FUNCTION_BLOCK FB_TimeLimitedIterator
VAR
    nLocalTaskUsagePercent : BYTE; 
    fbGetTickTime : GETCPUCOUNTER;
    TaskIndex : DINT;
    
    nInterruptThreshold : UDINT;
    nLocalCycleTime : UDINT;
    nIterationStartTime : ULINT;
    nIterationCurrentTime : ULINT;
    nIterationElapsedTime : UDINT;
END_VAR

METHOD PUBLIC CheckInterationTimeExceeded : BOOL
VAR_INPUT
END_VAR
fbGetTickTime();

nIterationCurrentTime := DWORD_TO_ULINT(fbGetTickTime.cpuCntLoDW) OR SHL(DWORD_TO_ULINT(fbGetTickTime.cpuCntHiDW), 32);
nIterationElapsedTime := ULINT_TO_UDINT (THIS^.nIterationCurrentTime - THIS^.nIterationStartTime);

CheckInterationTimeExceeded := nIterationElapsedTime >= nInterruptThreshold;
END_METHOD

METHOD CurrentIterationTime : LTIME
VAR
    CurrentTime : ULINT;
END_VAR
fbGetTickTime();

CurrentTime := DWORD_TO_ULINT(fbGetTickTime.cpuCntLoDW) OR SHL(DWORD_TO_ULINT(fbGetTickTime.cpuCntHiDW), 32);

CurrentIterationTime := ULINT_TO_LTIME (CurrentTime - THIS^.nIterationStartTime)*100;
END_METHOD

METHOD PUBLIC SetIterationStartTime : BOOL
VAR_INPUT
END_VAR
IF TaskIndex = 0 OR TaskIndex <> GETCURTASKINDEXEX() THEN
    TaskIndex := GETCURTASKINDEXEX();
    nLocalCycleTime := TwinCAT_SystemInfoVarList._TaskInfo[TaskIndex].CycleTime;
    nInterruptThreshold:= (nLocalCycleTime * LIMIT(1, TaskUsagePercent, 100)) / 100;
END_IF

fbGetTickTime();
nIterationStartTime := DWORD_TO_ULINT(fbGetTickTime.cpuCntLoDW) OR SHL(DWORD_TO_ULINT(fbGetTickTime.cpuCntHiDW), 32);
END_METHOD

PROPERTY PUBLIC TaskUsagePercent : BYTE
GET
TaskUsagePercent := nLocalTaskUsagePercent;
END_GET
SET
IF nLocalTaskUsagePercent <> TaskUsagePercent THEN
    nLocalTaskUsagePercent := TaskUsagePercent;
    
    TaskIndex := GETCURTASKINDEXEX();
	IF TaskIndex <> 0 THEN
		nLocalCycleTime := TwinCAT_SystemInfoVarList._TaskInfo[TaskIndex].CycleTime;
   	 	nInterruptThreshold:= (nLocalCycleTime * LIMIT(1, TaskUsagePercent, 100)) / 100;
	END_IF
END_IF
END_SET
END_PROPERTY

END_FUNCTION_BLOCK

(* stored: Version 1.1.0.1, ProductVersion 3.1.4024.12
   POU FB_TimeLimitedIterator: Id {feae5c23-357d-4ed9-9d1c-32ca973aa0ad}, SpecialFunc None
   Method CheckInterationTimeExceeded: Id {4a403e74-ab1f-4fc5-b865-65f6b1cbea9d}
   Method CurrentIterationTime: Id {ef19bc0c-ce47-460f-8ce7-bd21e0fb92be}
   Method SetIterationStartTime: Id {bc75f438-9ac1-4c8f-8351-10b88609b1b5}
   Property TaskUsagePercent: Id {633a7f1c-83a3-4054-9f1b-4b2eca7b9f45}
   Get Get: Id {a67d344e-d5c5-4c4d-a203-83178ed08983}
   Set Set: Id {6c064c68-a590-4d59-8175-798da213a006} *)
